FUNCTION_BLOCK TOffTimer
VAR
    TOF1 : TOF;
END_VAR

METHOD Delay : BOOL
VAR_INPUT
    In : BOOL;
END_VAR
TOF1(IN := In);
Delay := TOF1.Q;
END_METHOD

METHOD FB_init : BOOL
VAR_INPUT
	bInitRetains : BOOL; // if TRUE, the retain variables are initialized (warm start / cold start)
	bInCopyCode : BOOL;  // if TRUE, the instance afterwards gets moved into the copy code (online change)
    PresetTime : LREAL; // seconds
END_VAR
TOF1.PT := LREAL_TO_TIME(PresetTime * 1000);
END_METHOD

PROPERTY OutputState : BOOL
GET
OutputState := TOF1.Q;
END_GET
END_PROPERTY

PROPERTY PresetTime : LREAL
GET
PresetTime := TIME_TO_LREAL(TOF1.PT)/1000.0; // in seconds
END_GET
SET
TOF1.PT := LREAL_TO_TIME(PresetTime * 1000);
END_SET
END_PROPERTY

END_FUNCTION_BLOCK

(* stored: Version 1.1.0.1, ProductVersion 3.1.4024.3
   POU TOffTimer: Id {9b8fb8ef-b17f-4a39-93b3-d97e9d53661c}, SpecialFunc None
   Method Delay: Id {3ee9a384-9f47-4b54-8664-554515acf9cd}
   Method FB_init: Id {e089ed83-af93-4211-a099-8d5900bb900c}
   Property OutputState: Id {b4ce9aa4-0883-4bc8-8b64-1bb64747d61b}
   Get Get: Id {9cdb99fa-5849-40fa-9e35-86b5b51fb49b}
   Property PresetTime: Id {572b506d-ba56-4347-928c-4c78a3ef6cbe}
   Get Get: Id {d1147251-c67c-4112-9a51-df1726015dbd}
   Set Set: Id {8b33beac-0c53-4fe6-88bb-5181ff7449fa} *)
